(* Schneider Machine Expert - Basic project testHMI, file version 1.7.0.0 *)
(* ProjectInformations: Name=New project *)

HARDWARE
  Cpu 0: TM221ME16R/G
  EthernetConfiguration: NetworkName=M221, IpAllocationMode=FixedAddress, IpAddress=192.168.0.10, SubnetMask=255.255.255.0
  SerialLineConfiguration: Baud=Baud19200, Parity=ParityEven, DataBits=DataBits8, StopBits=StopBits1, PhysicalMedium=PhysicalMediumRs485, TransmissionMode=TransmissionModeModbusRtu, SlaveId=1, Addressing=SlaveAddressing
  MastTask: UsePeriodScanMode=false, PeriodScan=100
  FastTask: Period=255
  CpuBehavior: StartingMode=StartAsPreviousState, AutoSaveRamOnEeprom=true, WatchdogPeriod=250

SYMBOLS  (address, symbol, comment, settings)

POU New POU
  (* SectionNumber=0 *)

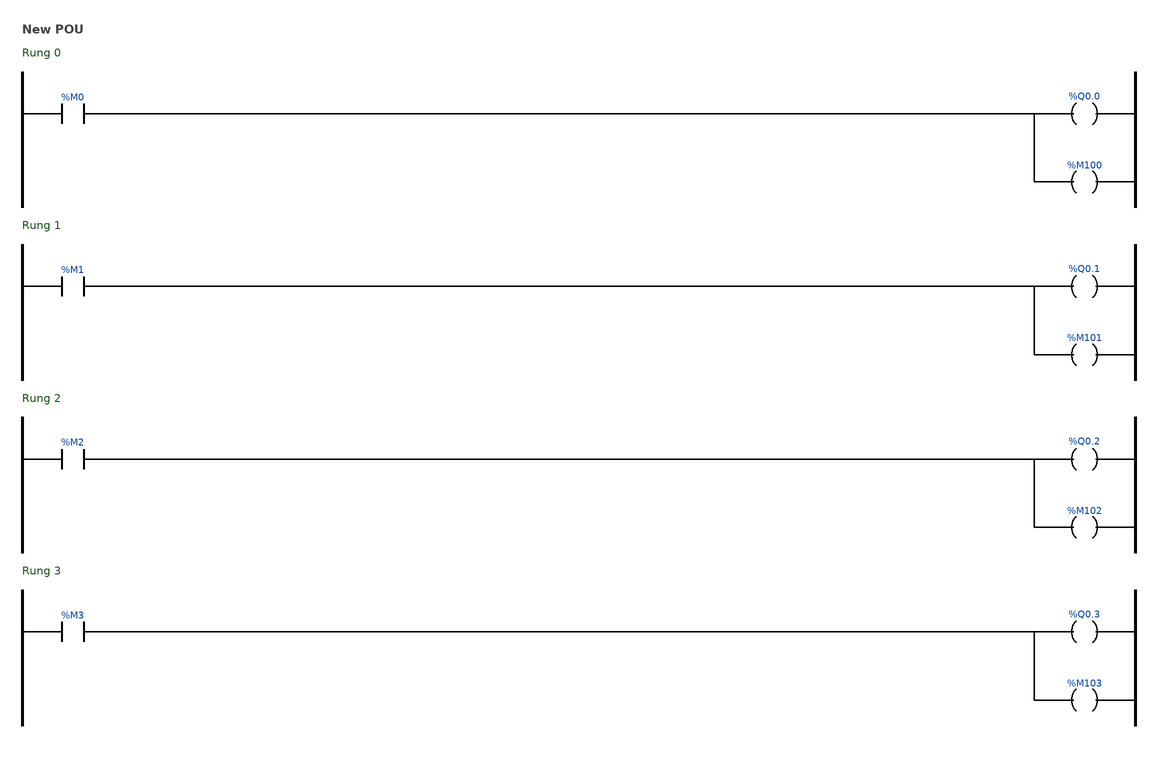

// Rung 0
  LD %M0
  ST %Q0.0
  ST %M100
  // as ST:
  //   %Q0.0 := %M0;
  //   %M100 := %M0;

// Rung 1
  LD %M1
  ST %Q0.1
  ST %M101
  // as ST:
  //   %Q0.1 := %M1;
  //   %M101 := %M1;

// Rung 2
  LD %M2
  ST %Q0.2
  ST %M102
  // as ST:
  //   %Q0.2 := %M2;
  //   %M102 := %M2;

// Rung 3
  LD %M3
  ST %Q0.3
  ST %M103
  // as ST:
  //   %Q0.3 := %M3;
  //   %M103 := %M3;

// Rung 4
  LD
